FUNCTION_BLOCK MotorTermFuse IMPLEMENTS I_TermFuse
VAR
	_input AT%I* :BOOL;
	
END_VAR

PROPERTY IsActive : BOOL
GET
IsActive := _input;
END_GET
END_PROPERTY

END_FUNCTION_BLOCK

(* stored: Version 1.1.0.1, ProductVersion 3.1.4024.12
   POU MotorTermFuse: Id {2bcfa7ff-b43c-4aa6-8d90-cefd9a2cbeb3}, SpecialFunc None
   Property IsActive: Id {db56a24f-5d66-4268-a71f-5e29406db3e4}
   Get Get: Id {7ce5753b-bc05-48a1-b2f2-c7db717ca361} *)
